PROGRAM MAIN
VAR
	tcpServer : TcpServer; 
END_VAR

tcpServer();

END_PROGRAM

(* stored: Version 1.1.0.1, ProductVersion 3.1.4018.2
   POU MAIN: Id {76d84d98-7320-4b96-b564-da36986ca222}, SpecialFunc None *)
